// TIA Portal V17 export
// export: Created 2025-06-26T07:49:38.311784Z, ExportSetting WithDefaults, DisplayName Totally Integrated Automation Portal, DisplayVersion V17 Update 8, DisplayName TIA Portal Openness, DisplayVersion V17 Update 8, DisplayName TIA Portal Version Control Interface, DisplayVersion V17, DisplayName STEP 7 Professional, DisplayVersion V17 Update 8, DisplayName STEP 7 Safety, DisplayVersion V17 Update 6, DisplayName WinCC Advanced, DisplayVersion V17 Update 8
FUNCTION_BLOCK "LubricationPriming"   // FB20, FBD
{ S7_Optimized_Access := 'TRUE' }
VERSION : 0.1
// stored: AutoNumber true, IsIECCheckEnabled false, IsRetainMemResEnabled false, MemoryReserve 100, SetENOAutomatically false, UDAEnableTagReadback false
   VAR_INPUT
      bEnable { ExternalAccessible := 'False'; ExternalVisible := 'False'; ExternalWritable := 'False'} : Bool;
      bReset { ExternalAccessible := 'False'; ExternalVisible := 'False'; ExternalWritable := 'False'} : Bool;
   END_VAR
   VAR
      Pump { ExternalAccessible := 'False'; ExternalVisible := 'False'; ExternalWritable := 'False'} : "fbOnOffRegulator";
      Special { S7_SetPoint := 'True'} : "fbSpecialRegulator";
   END_VAR
   VAR_TEMP
      bOutput : Bool;
   END_VAR
BEGIN

REGION Network 1: Pump regulator
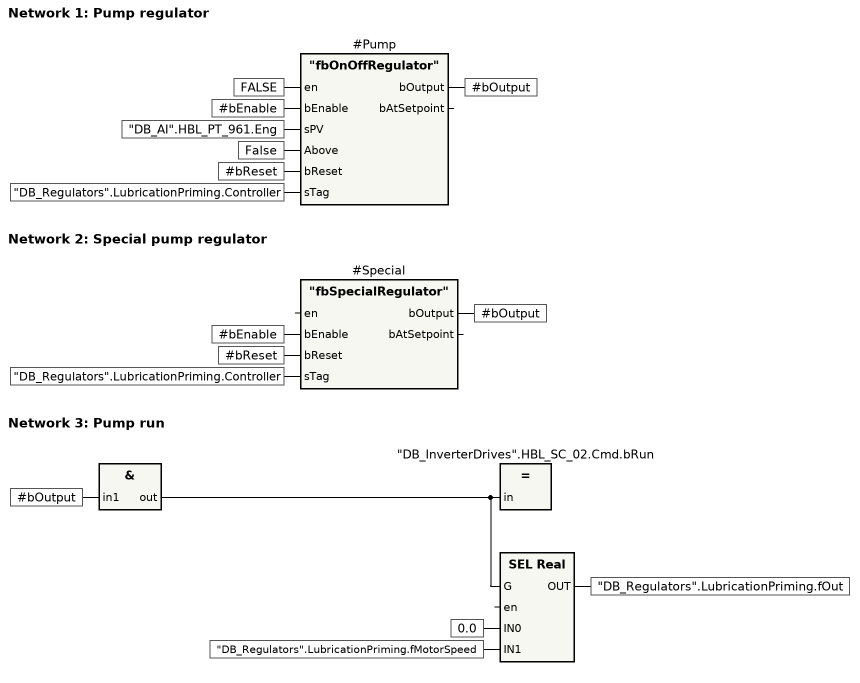
   IF FALSE THEN
       #Pump(bEnable := #bEnable,   // "fbOnOffRegulator"
             sPV := "DB_AI".HBL_PT_961.Eng,
             Above := False,
             bReset := #bReset,
             sTag := "DB_Regulators".LubricationPriming.Controller,
             bOutput => #bOutput);
   END_IF;
END_REGION

REGION Network 2: Special pump regulator
   // ##TEST: special situations require special regulators!
   #Special(bEnable := #bEnable,   // "fbSpecialRegulator"
            bReset := #bReset,
            sTag := "DB_Regulators".LubricationPriming.Controller,
            bOutput => #bOutput);
END_REGION

REGION Network 3: Pump run
   "DB_InverterDrives".HBL_SC_02.Cmd.bRun := #bOutput;
   "DB_Regulators".LubricationPriming.fOut := SEL(G := #bOutput, IN0 := 0.0, IN1 := "DB_Regulators".LubricationPriming.fMotorSpeed);
END_REGION

REGION Network 4: Inverter run
END_REGION
END_FUNCTION_BLOCK
